SUBAPPLICATION Uebung_038 (* Lauflicht 8 reine Zeitsteuerung *)
  (* Standard: 61499-2; Description: Copyright (c) 2023 Meisterschulen am Ostbahnhof This program and the accompanying materials are made available under the terms of the Eclipse Public License 2.0 which is available at https://www.eclipse.org/legal/epl-2.0/ SPDX-License-Identifier: EPL-2.0 *)
  (* Version 1.0, 2023-10-23, Franz Höpfinger, Meisterschulen am Ostbahnhof *)
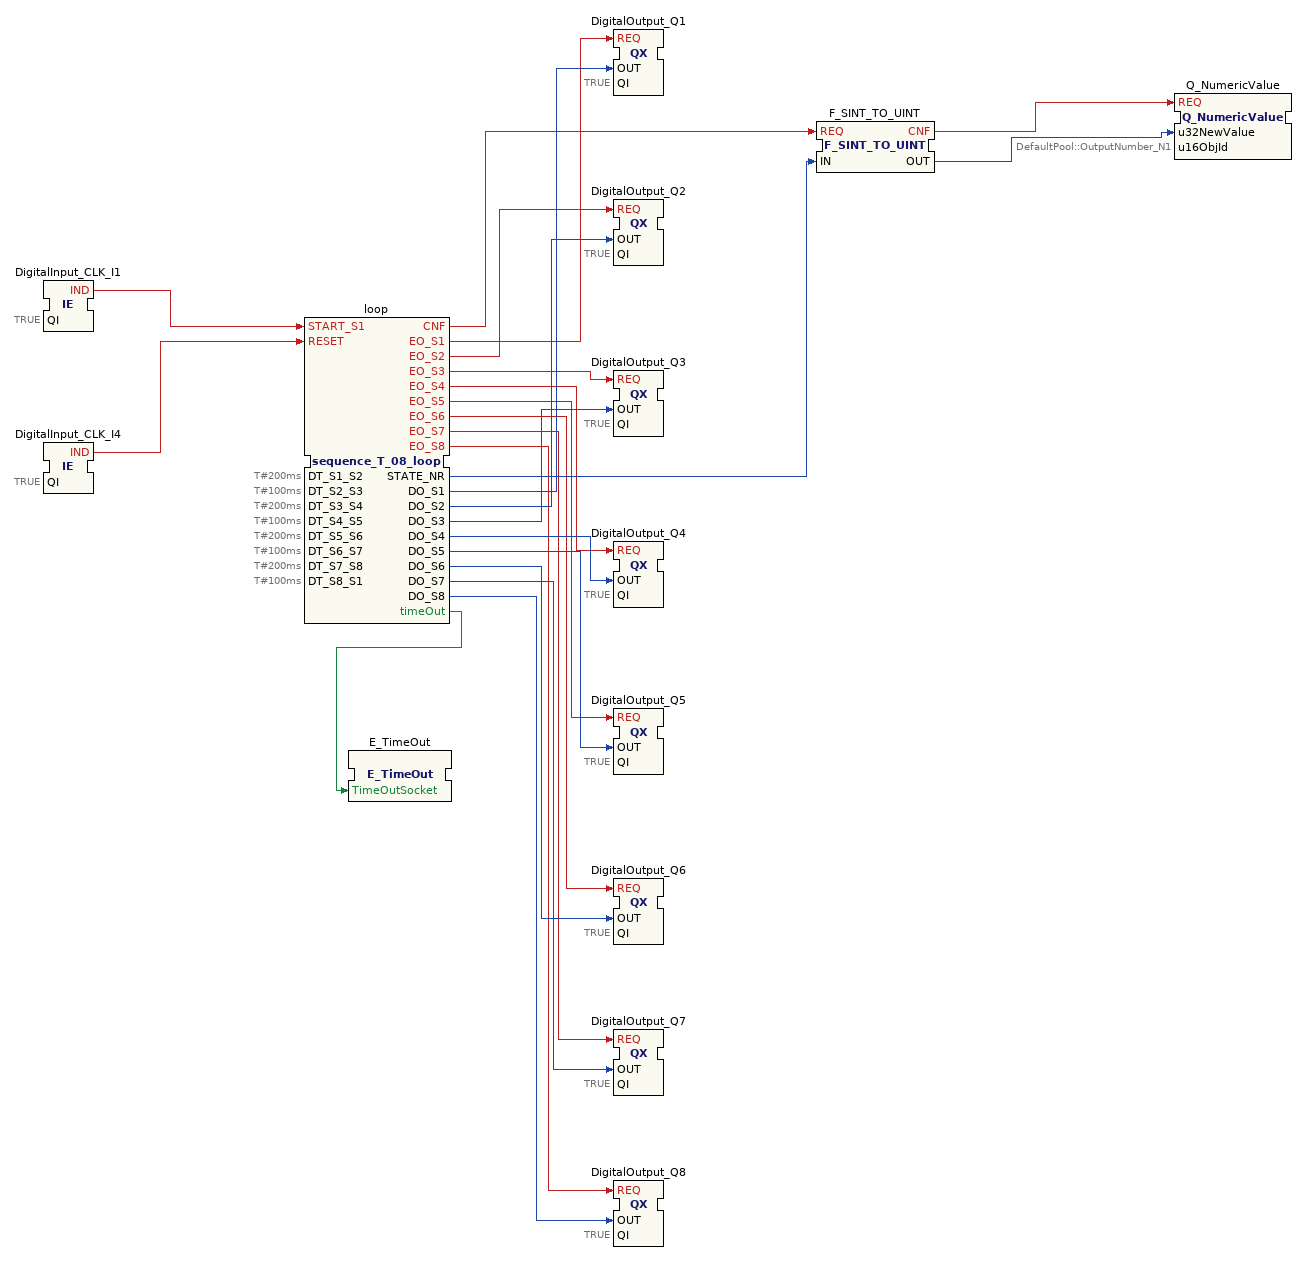
  FBS
    DigitalOutput_Q1 : QX(QI := TRUE);
    E_TimeOut : E_TimeOut;
    DigitalOutput_Q2 : QX(QI := TRUE);
    DigitalOutput_Q3 : QX(QI := TRUE);
    DigitalOutput_Q4 : QX(QI := TRUE);
    DigitalInput_CLK_I1 : IE(QI := TRUE);
    DigitalInput_CLK_I4 : IE(QI := TRUE);
    DigitalOutput_Q5 : QX(QI := TRUE);
    DigitalOutput_Q6 : QX(QI := TRUE);
    DigitalOutput_Q7 : QX(QI := TRUE);
    DigitalOutput_Q8 : QX(QI := TRUE);
    Q_NumericValue : Q_NumericValue(u16ObjId := DefaultPool::OutputNumber_N1);
    F_SINT_TO_UINT : F_SINT_TO_UINT;
    loop : sequence_T_08_loop(DT_S1_S2 := T#200ms, DT_S2_S3 := T#100ms, DT_S3_S4 := T#200ms, DT_S4_S5 := T#100ms, DT_S5_S6 := T#200ms, DT_S6_S7 := T#100ms, DT_S7_S8 := T#200ms, DT_S8_S1 := T#100ms);
  END_FBS
  EVENT_CONNECTIONS
    F_SINT_TO_UINT.CNF TO Q_NumericValue.REQ;
    DigitalInput_CLK_I1.IND TO loop.START_S1;
    DigitalInput_CLK_I4.IND TO loop.RESET;
    loop.CNF TO F_SINT_TO_UINT.REQ;
    loop.EO_S1 TO DigitalOutput_Q1.REQ;
    loop.EO_S2 TO DigitalOutput_Q2.REQ;
    loop.EO_S3 TO DigitalOutput_Q3.REQ;
    loop.EO_S4 TO DigitalOutput_Q4.REQ;
    loop.EO_S5 TO DigitalOutput_Q5.REQ;
    loop.EO_S6 TO DigitalOutput_Q6.REQ;
    loop.EO_S7 TO DigitalOutput_Q7.REQ;
    loop.EO_S8 TO DigitalOutput_Q8.REQ;
  END_CONNECTIONS
  DATA_CONNECTIONS
    F_SINT_TO_UINT.OUT TO Q_NumericValue.u32NewValue;
    loop.STATE_NR TO F_SINT_TO_UINT.IN;
    loop.DO_S1 TO DigitalOutput_Q1.OUT;
    loop.DO_S2 TO DigitalOutput_Q2.OUT;
    loop.DO_S3 TO DigitalOutput_Q3.OUT;
    loop.DO_S4 TO DigitalOutput_Q4.OUT;
    loop.DO_S5 TO DigitalOutput_Q5.OUT;
    loop.DO_S6 TO DigitalOutput_Q6.OUT;
    loop.DO_S7 TO DigitalOutput_Q7.OUT;
    loop.DO_S8 TO DigitalOutput_Q8.OUT;
  END_CONNECTIONS
  ADAPTER_CONNECTIONS
    loop.timeOut TO E_TimeOut.TimeOutSocket;
  END_CONNECTIONS
END_SUBAPPLICATION
